// TIA Portal project "TIA-Prgm-ATV320-rv3" (V15.1)

(* hardware
DEVICE "GSD device_1"  GSD.Device.PN
   slot 0: "ATV320"  ATV320  ATV320
      slot 0: "ATV320"  ATV320
      slot 1: "Interface"  Interface
         slot 1: "Port 1"  Port 1
         slot 2: "Port 2"  Port 2
   slot 0: "Rack"  Rack  V1.0
   slot 1: "Telegram 101 (4PKW/6PZD)_1"  Telegram 101 (4PKW/6PZD)
      slot 0: "Telegram 101"  Telegram 101
DEVICE "S7-1200 station_1"  S7-1200 Station
   slot 0: "Rack_0"  S7-1200 Rack  Rack  V1.0
   slot 1: "PLC_1"  CPU 1215C DC/DC/DC  6ES7 215-1AG40-0XB0  V4.0
*)

// ===== PLC "PLC_1"  CPU 1215C DC/DC/DC =====
// protected blocks, not shown: "ATV320_rv3"

VAR_GLOBAL   // PLC tag table "VFD_Tag_List"
   "Amps_In" AT %IW82 : UInt;   // Amps feedback from drive
   "Amps_Out" AT %MD0 : Real;
   "Ctrl_Word" AT %QW76 : Word;   // Command word to drive
   "E_Stop" AT %M0.5 : Bool;
   "Enable" AT %M0.3 : Bool;
   "Fault_Code" AT %IW84 : Word;   // Fault code from drive
   "Freq_Fdbk_In" AT %IW86 : Word;   // Frequency feedback from drive
   "Line_Volts_In" AT %IW80 : UInt;   // Line voltage reading from drive
   "Motor_Rpms_In" AT %IW78 : Int;   // Here if you need it. Not in this block
   "Reset_Fault" AT %M0.2 : Bool;
   "Run_Fwd" AT %M0.0 : Bool;
   "Run_Rev" AT %M0.1 : Bool;
   "Speed_Out_Hz" AT %QW78 : Int;   // Output Speed setpoint to Drive.
   "Speed_Setpoint_Hz" AT %MD4 : Real;   // Set desired speed in Hz `00.0Hz to 60.0Hz`
   "Status_Word" AT %IW76 : Word;   // Drive Status Word
   "Stop" AT %M0.4 : Bool;
END_VAR

ORGANIZATION_BLOCK "Main"   // OB1, LAD, ProgramCycle
TITLE = "Main Program Sweep (Cycle)"
{ S7_Optimized_Access := 'TRUE' }
VERSION : 0.1
   VAR_INPUT
      Initial_Call : Bool;   // Initial call of this OB
      Remanence : Bool;   // =True, if remanent data are available
   END_VAR
BEGIN

REGION Network 1
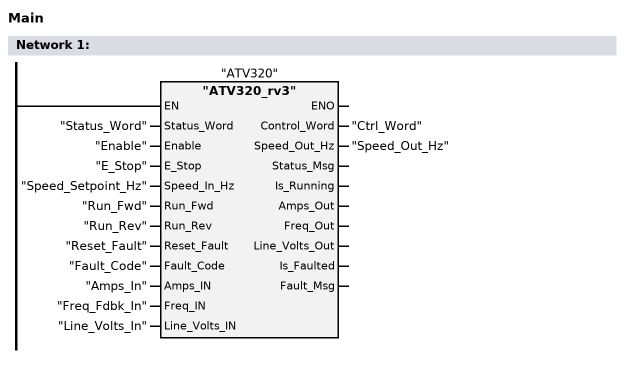
   RUNG wire#powerrail
      "ATV320"(Status_Word := "Status_Word", Enable := "Enable", E_Stop := "E_Stop", Speed_In_Hz := "Speed_Setpoint_Hz", Run_Fwd := "Run_Fwd", Run_Rev := "Run_Rev", Reset_Fault := "Reset_Fault", Fault_Code := "Fault_Code", Amps_IN := "Amps_In", Freq_IN := "Freq_Fdbk_In", Line_Volts_IN := "Line_Volts_In", Control_Word => "Ctrl_Word", Speed_Out_Hz => "Speed_Out_Hz", Status_Msg =>, Is_Running =>, Amps_Out =>, Freq_Out =>, Line_Volts_Out =>, Is_Faulted =>, Fault_Msg =>)
   END_RUNG
   // the same network as SCL:
   "ATV320"(Status_Word := "Status_Word",   // "ATV320_rv3"
            Enable := "Enable",
            E_Stop := "E_Stop",
            Speed_In_Hz := "Speed_Setpoint_Hz",
            Run_Fwd := "Run_Fwd",
            Run_Rev := "Run_Rev",
            Reset_Fault := "Reset_Fault",
            Fault_Code := "Fault_Code",
            Amps_IN := "Amps_In",
            Freq_IN := "Freq_Fdbk_In",
            Line_Volts_IN := "Line_Volts_In",
            Control_Word => "Ctrl_Word",
            Speed_Out_Hz => "Speed_Out_Hz");
END_REGION
END_ORGANIZATION_BLOCK